Staubli VAL3: ISO_PDU_DATA_T.pjx

Parameters version=s7.9.1 stackSize=5000 millimeterUnit=true
Data file=ISO_PDU_DATA_T.dtx
Type name=S7telegram_T path=./S7telegram_T/S7telegram_T.pjx
